TYPE ST_LaudaReadCommands_Pump :
STRUCT
	FlowRate	: STRING := 'IN_PV_07';
	PowerStage	: STRING := 'IN_SP_01';
END_STRUCT
END_TYPE

(* stored: Version 1.1.0.1, ProductVersion 3.1.4024.13
   DUT ST_LaudaReadCommands_Pump: Id {7bd00d58-b29d-4c60-b629-8bdb686bb81c} *)
